Xinje XDPPro project, PLC1: XL5E-16 (software 3.7.14b 2022-06-24)

PROGRAM 梯形图

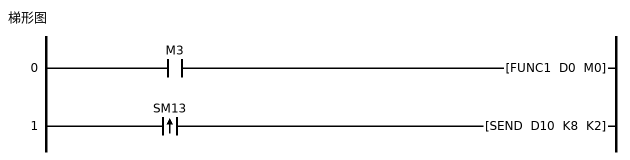
LD     M3
FUNC1  D0 M0
LDP    SM13
SEND   D10 K8 K2

C FUNCTION BLOCK func1.fcb
/* #EXPORT_ENTRY_BEGIN(FUNC1)
//    类型              模式             个数               映射          注释
W = { type = "PINT16S", mode = [In,Out], count = "unknown", map = [D,HD], comment = "" }
B = { type = "BIT"    , mode = [In,Out], count = "unknown", map = [M,HM], comment = "" }
#EXPORT_ENTRY_END */
/*************************************************************************
 * FunctionBlockName:  FUNC1
 * Version:            1.0.0
 * Author:             
 * UpdateTime:         2022-10-12 10:03:59
 * Comment:            
**************************************************************************/

/**
 * @summary 
 * @param W 
 * @param B 
 */
void FUNC1(PINT16S W,BIT B)
{
	#define SysRegAddr_HD_D_HM_M
    D[10] = 0X94;
    D[11] = 0X01;
    D[12] = 0X64;
    D[13] = 0X00;
    D[14] = 0X6E;
    D[15] = 0x4C;
    D[16] = 0x32;
    D[17] = 0x75;
}